PROGRAM V0_10
VAR
END_VAR

(*
	Twee Pompen
	
	Een tank wordt gevuld met twee pompen. Om onderhoud te vermijden en de slijtage aan de pompen te spreiden zal men elke pomp om beurten apart laten werken. De installatie zal pas werken als een hoofdschakelaar AAN staat.

	De pompbeweging wordt gestart ofwel:
    	manueel door een startdrukknop
    	automatisch door een niveauschakelaar (onderin de tank)

	De pompbeweging wordt gestopt ofwel:
    	manueel door een stopdrukknop
    	automatisch door een niveauschakelaar (bovenaan de tank)
*)

END_PROGRAM

(* stored: Version 1.1.0.1, ProductVersion 3.1.4024.12
   POU V0_10: Id {354420ea-f2ab-4e38-ad43-bba07bd01c98}, SpecialFunc None *)
